(* Logix 5000 project; controller Services vendor 1 type 14 code 77 rev 16.21; software revision 16.03 *)

TASK MainTask (continuous, watchdog 500 ms) : MainProgram

MODULES
   Controller : vendor 1 type 14 code 77 (CompactLogixL32EController 0, rev 16.21)
      LocalENB : 1769-L32E Ethernet Port (CompactLogixL32Ethernet 1, rev 16.3)
      Local : CompactBus (CompactVirtualAdapter 3, rev 16.3, Input RPI 5 ms)
          : 1769-IQ16 (Compact 3, rev 1.1, Input RPI 20 ms)
          : 1769-IQ16 (Compact 4, rev 1.1, Input RPI 20 ms)
          : vendor 1 type 10 code 33 (Compact 6, rev 1.1, Output RPI 5 ms)
          : vendor 1 type 10 code 33 (Compact 1, rev 1.1, Output RPI 5 ms)
          : 1769-OB16P (Compact 2, rev 2.1, Output RPI 20 ms)
          : 1769-OB16P (Compact 5, rev 2.1, Output RPI 20 ms)
END_MODULES

VAR_GLOBAL   (* controller tags *)
   L1 : DINT;
   L2 : DINT;
   L4 : DINT;
   N4 : DINT;
   Timer1 : TIMER := (PRE := 2000, ACC := 79, EN := 1, TT := 1);
   timer2 : TIMER := (PRE := 8000);
   X : DINT[130] := ([0] := 16385, [1] := 321, [2] := 128, [3] := 32, [4] := 4993, [5] := 4993, [8] := 15, [9] := 32744, [10] := 21616, [11] := 9600, [12] := 32744, [13] := 8, [14] := 8, [15] := 8, [16] := 8, [17] := 1, [18] := 1, [19] := 10256, [20] := 10120, [27] := 1, [28] := 8, [30] := 8, [31] := 8, [32] := 8, [45] := 7, [46] := 25056, [47] := 9416, [48] := 10184, [49] := 9992, [50] := 10136, [51] := 10160, [52] := 8, [54] := 1, [56] := 6608, [57] := 9936, [58] := 6264, [59] := 8, [60] := 8, [61] := 6248, [62] := 8, [64] := 16, [65] := 16, [66] := 8, [67] := 8, [73] := 71, [74] := 32744, [75] := 32736, [76] := 25736, [77] := 8, [78] := 8464, [79] := 7656, [80] := 104, [81] := 7296, [82] := 7440, [83] := 7264, [84] := 7200, [85] := 7240, [86] := 1, [87] := 8, [88] := 6112,
        [89] := 6104, [90] := 8, [91] := 6288, [95] := 8, [96] := 8, [97] := 16, [98] := 8, [99] := 85, [100] := 16, [104] := 373, [105] := 68, [106] := 8, [107] := 9808, [108] := 8744, [109] := 8, [110] := 9632, [111] := 9632, [112] := 9152, [113] := 9288);
        [1]   // OUTLET TEMPERATURE
        [4]   // INSIDE PRESSURE
        [0]   // INLET TEMPERATURE
        [2]   // CONDENSER TEMPERATURE
        [7]   // DINP 17 - 20
        [3]   // FAN CURRENT
        [5]   // OUTSIDE PRESSURE
        [6]   // DINP 1 - 16
   Y : DINT[40] := ([0] := 1, [33] := 2);
END_VAR

PROGRAM MainProgram   (* main routine MainRoutine *)

ROUTINE MainRoutine   (* ladder *)
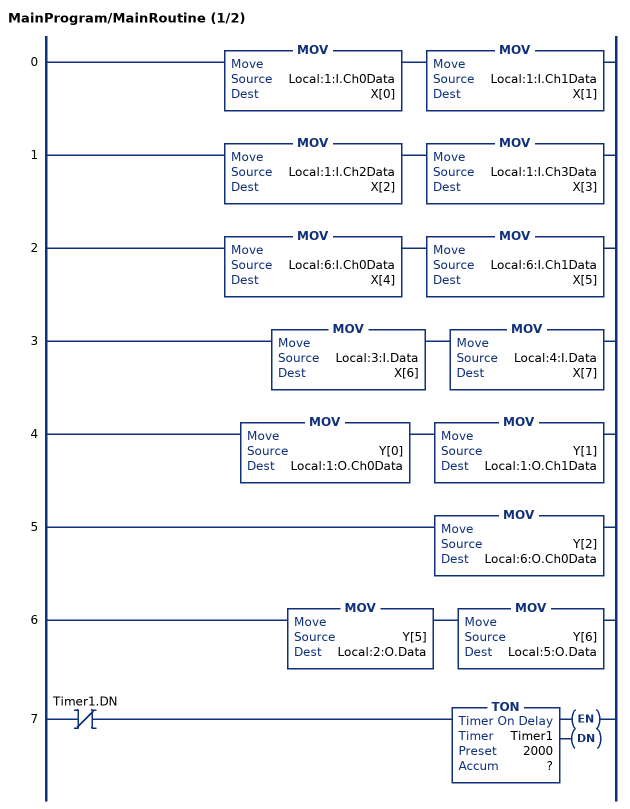
   0: MOV(Local:1:I.Ch0Data,X[0])MOV(Local:1:I.Ch1Data,X[1]);
   1: MOV(Local:1:I.Ch2Data,X[2])MOV(Local:1:I.Ch3Data,X[3]);
   2: MOV(Local:6:I.Ch0Data,X[4])MOV(Local:6:I.Ch1Data,X[5]);
   3: MOV(Local:3:I.Data,X[6])MOV(Local:4:I.Data,X[7]);
   4: MOV(Y[0],Local:1:O.Ch0Data)MOV(Y[1],Local:1:O.Ch1Data);
   5: MOV(Y[2],Local:6:O.Ch0Data);
   6: MOV(Y[5],Local:2:O.Data)MOV(Y[6],Local:5:O.Data);
   7: XIO(Timer1.DN)TON(Timer1,?,?);
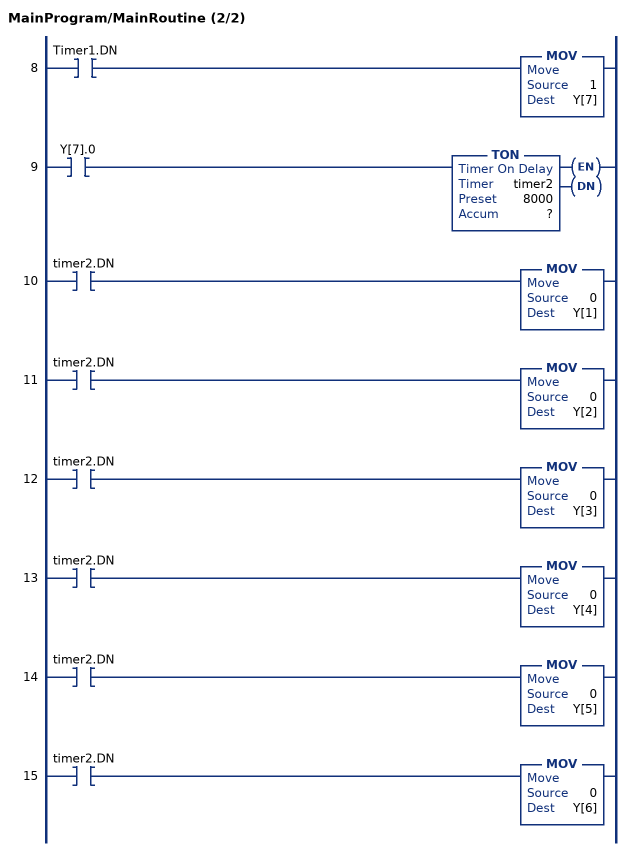
   8: XIC(Timer1.DN)MOV(1,Y[7]);
   9: XIC(Y[7].0)TON(timer2,?,?);
   10: XIC(timer2.DN)MOV(0,Y[1]);
   11: XIC(timer2.DN)MOV(0,Y[2]);
   12: XIC(timer2.DN)MOV(0,Y[3]);
   13: XIC(timer2.DN)MOV(0,Y[4]);
   14: XIC(timer2.DN)MOV(0,Y[5]);
   15: XIC(timer2.DN)MOV(0,Y[6]);
END_ROUTINE
END_PROGRAM
